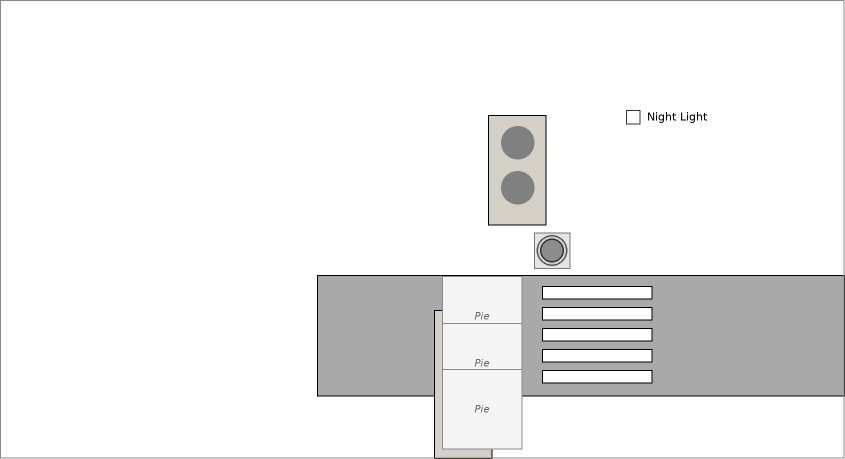
VISUALIZATION Visualization  // 845x459
    PushSwitch (534,232 36x37), variable: GVL.StartButton, behaviour: TAP, style: Switch-PushSwitch-Gray
    Rectangle (317,275 528x121)
    Checkbox (624,102 111x30), "Night Light", variable: GVL.NightLight
    Rectangle (542,286 110x13)
    Rectangle (542,307 110x13)
    Rectangle (542,328 110x13)
    Rectangle (542,349 110x13)
    Rectangle (542,370 110x13)
    Rectangle (488,115 58x110)
    Ellipse (500,125 35x35), colour toggle: GVL.CrossWalkRedLight
    Ellipse (500,170 35x35), colour toggle: GVL.CrossWalkGreenLight
    Rectangle (434,310 58x149)
    Pie (442,276 80x80), colour toggle: GVL.CarRedLight
    Pie (442,323 80x80), colour toggle: GVL.CarYellowLight
    Pie (442,369 80x80), colour toggle: GVL.CarGreenLight
END_VISUALIZATION

(* stored: Version 1.1.0.1, ProductVersion 3.1.4024.15
   Visu Visualization: Id {455ebbfe-c397-45c6-b3e9-2b571a4b5bbf} *)
